PROGRAM BundleToJson
VAR
	fbJson : FB_JsonSaxWriter;
	fbJsonDataType : FB_JsonReadWriteDataType;
	jsonDoc : STRING(100000); //this wont even show up in online view as twincat cannot show strings this long
	arrDoc : ARRAY[0..100000] OF BYTE;
	
	newBundle : Bundle;
	getBundle : Bundle;
END_VAR

newBundle.id := 'abcdefghijkl';
newBundle.autoRE := TRUE;
newBundle.cardboard := MAIN.moduleA22.materialsArr;
newBundle.timeDone := MAIN.currentTime;

fbJson.ResetDocument();
fbJsonDataType.AddJsonValueFromSymbol(fbJson, 'Bundle', SIZEOF(newBundle), ADR(newBundle));
fbJson.CopyDocument(jsonDoc, SIZEOF(jsonDoc));

MEMCPY(
	ADR(arrDoc), 
	ADR(jsonDoc),
	MIN(
		SIZEOF(jsonDoc),
		SIZEOF(arrDoc))
	);
	
fbJsonDataType.SetSymbolFromJson(jsonDoc, 'Bundle', SIZEOF(getBundle), ADR(getBundle));

END_PROGRAM

(* stored: Version 1.1.0.1, ProductVersion 3.1.4024.11
   POU BundleToJson: Id {f60b91ab-2049-43d9-a925-115cd4098610}, SpecialFunc None *)
